// TwinCAT 3 PLC project PMPS
// Title: PMPS
// Company: SLAC - LCLS
// Author: Alex Wallace and contributors
// ProjectVersion: 0.0.0
// Description: Collection of PMPS functionality for LCLS PLCs
// ProgramVersion: 3.1.4023.0
// CompilerDefines: L
// libraries:
//   LCLS General, * (SLAC)
//   Tc2_MC2, * (Beckhoff Automation GmbH)
//   Tc2_Standard, * (Beckhoff Automation GmbH)
//   Tc2_System, * (Beckhoff Automation GmbH)
//   Tc2_Utilities, * (Beckhoff Automation GmbH)
//   Tc3_JsonXml, * (Beckhoff Automation GmbH)
//   Tc3_Module, * (Beckhoff Automation GmbH)
//   TcUnit,1.2.0.0,www.tcunit.org
// project tree:
//   AncillaryComponents/ FB_JsonDocToSafeBP.TcPOU, FB_JsonFileToJsonDoc.TcPOU (not stored), FB_TempSensor_FFO.TcPOU (not stored), FB_PressSensor_FFO.TcPOU (not stored)
//   DUTs/InternalDUT/ E_MPSBeamRates.TcDUT (not stored), E_MPSBeamClasses.TcDUT (not stored), K_Apertures.TcDUT (not stored), K_Attenuators.TcDUT (not stored), K_Stopper.TcDUT, L_Apertures.TcDUT (not stored), L_Attenuators.TcDUT (not stored), L_Stopper.TcDUT (not stored), ST_AttenuatorStatus.TcDUT (not stored), ST_BP_ArbInternal.TcDUT (not stored), ST_FF.TcDUT (not stored), ST_FFInfo.TcDUT (not stored), ST_FFOverride.TcDUT (not stored), ST_PMPS_Aperture.TcDUT (not stored), ST_PMPS_Attenuator.TcDUT (not stored), T_HashTableEntry.TcDUT (not stored)
//   DUTs/ PMPS_CODES.TcDUT (not stored), ST_DeviceState.TcDUT (not stored), ST_DeviceStateExt.TcDUT (not stored), ST_DeviceStateTable.TcDUT (not stored)
//   DUTs/UserDUT/ E_BridgeLinkStatus.TcDUT (not stored), E_BridgeStatus.TcDUT (not stored), E_DataStatus.TcDUT (not stored), E_EcCommState.TcDUT (not stored), ST_ReactiveParams.TcDUT (not stored), ST_BeamParams.TcDUT (not stored), ST_DbStateParams.TcDUT (not stored), ST_Device.TcDUT (not stored)
//   GVLs/ PMPS_GVL.TcGVL (not stored), PMPS_PARAM.TcGVL, PMPS_TOOLS.TcGVL (not stored)
//   HelperFunctions/ FB_DummyHA.TcPOU (not stored), FB_DummyArbIO.TcPOU (not stored), F_BPWithID.TcPOU (not stored), F_DifferentBeamParams.TcPOU (not stored), F_eVExcludeRange.TcPOU (not stored), F_eVIncludeRange.TcPOU (not stored), F_eVRangeCalculator.TcPOU (not stored), F_eVWithinSpec.TcPOU (not stored), F_InitTestBP.TcPOU (not stored), F_SafeBPCompare.TcPOU (not stored), F_SafeBPCompare0Rate.TcPOU (not stored), F_SetBeamParams.TcPOU (not stored), F_SetGoodAttStatus.TcPOU (not stored), F_SetStateParams.TcPOU (not stored), F_PMPS_JSON.TcPOU (not stored), F_ValidReqID.TcPOU (not stored), PE_Ranges.TcPOU (not stored), F_AttenuatorOK.TcPOU (not stored)
//   HelperFunctions/TypeTranslators/ APT_TO_IO.TcPOU (not stored), ATT_TO_IO.TcPOU (not stored), BP_TO_IO.TcPOU (not stored), F_DeviceState_To_DeviceStateExt.TcPOU (not stored), IO_TO_APT.TcPOU (not stored), IO_TO_ATT.TcPOU (not stored), IO_TO_BP.TcPOU (not stored)
//   ImplicitChecks/ CheckBounds.TcPOU (not stored), CheckDivDInt.TcPOU (not stored), CheckDivLInt.TcPOU (not stored), CheckDivLReal.TcPOU (not stored), CheckDivReal.TcPOU (not stored), CheckLRangeSigned.TcPOU (not stored), CheckLRangeUnsigned.TcPOU (not stored), CheckPointer.TcPOU (not stored), CheckRangeSigned.TcPOU (not stored), CheckRangeUnsigned.TcPOU (not stored)
//   / MAIN.TcPOU (not stored), PlcTask.TcTTO (not stored)
//   MajorComponents/Arbiter/ FB_VetoArbiter.TcPOU (not stored), FB_Arbiter.TcPOU (not stored), FB_BeamParamAssertionPool.TcPOU (not stored)
//   MajorComponents/BPTM/ BeamParameterTransitionManager.TcPOU (not stored), E_BPTMState.TcDUT (not stored)
//   MajorComponents/ FB_BPControlDevice.TcPOU (not stored), FB_RateFromEPICS.TcPOU (not stored), FB_BeamClassFromEPICS.TcPOU (not stored), I_LowerAuthority.TcIO (not stored), I_UndulatorComplex.TcIO (not stored), FB_BPRequestor.TcPOU (not stored), FB_LinearDeviceStateTable.TcPOU (not stored), FB_LinearGovernor.TcPOU (not stored), I_HigherAuthority.TcIO (not stored)
//   MajorComponents/PhotonEnergyInterface/ FB_AcceleratorLinks.TcPOU (not stored), FB_Hgvpu.TcPOU (not stored), FB_LPhotonEnergy.TcPOU (not stored), FB_KPhotonEnergy.TcPOU (not stored), FB_PhotonEnergy.TcPOU (not stored), FB_SXU.TcPOU, FB_UndulatorSegment.TcPOU (not stored), F_CalculatePhotonEnergy.TcPOU (not stored)
//   MajorComponents/FastFaults/ FB_FastFault.TcPOU (not stored), FB_HardwareFFOutput.TcPOU
//   MajorComponents/InterPlcComm/ FB_ArbiterToSubSys_IO.TcPOU, FB_BridgeDiagnostics.TcPOU (not stored), FB_SubSysToArbiter_IO.TcPOU (not stored)
//   MajorComponents/InterPlcComm/Sanitization/ I_FallibleLreal.TcIO (not stored), FB_FallibleRealFromEtherCAT.TcPOU (not stored)
//   MajorComponents/PMPS_MPS_Interface/ FB_BeamClassOutputs.TcPOU (not stored), FB_BeamClassOutputs_BCD.TcPOU (not stored), FB_CTLS_Outputs.TcPOU (not stored), FB_MachineModeFromEPICS.TcPOU (not stored), FB_PhotonEnergyWatcher.TcPOU (not stored), FB_BeamClassWatcher.TcPOU (not stored)
//   MajorComponents/SimulationFB/ FB_eVSimulator.TcPOU (not stored), FB_MachineSimulator.TcPOU (not stored)
//   MajorComponents/Stoppers/ FB_KStopper.TcPOU (not stored), FB_KVetoDevice.TcPOU (not stored), FB_LVetoDevice.TcPOU (not stored), FB_LStopper.TcPOU (not stored), FB_StopperWatcher.TcPOU (not stored), FB_VetoDevice.TcPOU (not stored)
//   TestComponents/DUT/ E_ArbDosTestStates.TcDUT (not stored), E_BPTMTestStates.TcDUT (not stored)
//   TestComponents/ FB_Arbiter_Test.TcPOU (not stored), FB_VetoArbiter_Test.TcPOU (not stored), FB_AttenuatorSimulator.TcPOU (not stored), FB_BPTM_Test.TcPOU (not stored), FB_ArbToSubsys_Test.TcPOU (not stored), FB_DiffBP_Test.TcPOU (not stored), FB_SubsysToArb_Test.TcPOU (not stored), FB_evRangeCalculator_Test.TcPOU (not stored), FB_eVWithinSpec_Test.TcPOU (not stored), FB_FastFault_Test.TcPOU (not stored), FB_PhotonEnergyWatcher_Test.TcPOU (not stored), FB_SafeBPCompare_Test.TcPOU (not stored), FB_SolidAttenuator.TcPOU (not stored) (excluded from build)

// ---- DUTs/InternalDUT/K_Stopper.TcDUT
{attribute 'qualified_only'}
{attribute 'strict'}
TYPE K_Stopper :
(
    ST3K4 := 1, // TMO PPS stopper in
    ST1K2 := 2, // RIX PPS stopper in
    MR1K1_IN := 3, // Monochromator focus optic vertical state
    MR1K1_OUT := 4, // Monochromator focus optic vertical state
    MR1K3_IN := 5, // TXI MR1K3 Offset Mirror horizontal state
    MR1K3_OUT := 6, // TXI MR1K3 Offset Mirror horizontal state
    ST4K4 := 7, //TMO ST4K4 Photon Terminator In Limit Switch
    ST1K0 := 8, //Test Photon Stopper in the FEE
    ST1K3 :=9, //TXI Kline PPS stopper in
    MR2K3_IN := 10, // TXI MR2K3 Offset Mirror state
    MR2K3_OUT := 11, // TXI MR2K3 Offset Mirror horizontal state
    DEFAULT := PMPS_GVL.MAX_VETO_DEVICES // DO NOT USE FOR ANYTHING
);
END_TYPE

// ---- GVLs/PMPS_PARAM.TcGVL
{attribute 'qualified_only'}
VAR_GLOBAL CONSTANT
    MAX_FAST_FAULTS	:	UINT := 50; // Max fast faults for an FFO
    MAX_ASSERTIONS    :    UDINT := 20; //Maximum number of BP requests in the arbiter
    TRANS_MARGIN : REAL := REAL#0.05; // Allowed % margin above requested transmission level in SafeBPCompare (0.0500 = 5deci% default). Note: change this value if scaling factor changes.
END_VAR

// ---- AncillaryComponents/FB_JsonDocToSafeBP.TcPOU
FUNCTION_BLOCK FB_JsonDocToSafeBP
VAR_INPUT
	bExecute             : BOOL; //Rising Edge
	jsonDoc 		: SJsonValue;
	sDeviceName : STRING;
END_VAR
VAR_OUTPUT
	bHasDevice		: BOOL;
	bHasAllStates		: BOOL;
	bHasAllParameters :BOOL := TRUE;
	bBusy                : BOOL;
    bError               : BOOL;
    nErrId               : UDINT;
	sErrMsg				 :STRING;
END_VAR
VAR_IN_OUT
	arrStates: ARRAY[*] OF ST_DbStateParams;
	io_fbFFHWO    :    FB_HardwareFFOutput;
END_VAR
VAR
	(* JSON *)
	fbJson 			: FB_JsonDomParser;
	jsonProp		: SJsonValue;
	jsonValue		: SJsonValue;
	jsonParam		: SJsonValue;
	jsonnTran      : SJsonValue;
	jsonnRate      : SJsonValue;
	Step: INT;
	index: DINT;
	nStateCount:DINT;
    RisingEdge           : R_TRIG;

	(*Logger*)
	tNewMessage : R_TRIG;
    fbLogger : FB_LogMessage := (eSubsystem:=E_SubSystem.MPS, nMinTimeViolationAcceptable:=10);	
	(*FFO*)
	FFO    :    FB_FastFault :=(
        i_Desc := 'Fault occurs when there is an error loading safe beam parameters from json file',
        i_TypeCode := 16#FF13);
	sbuffReadSmall: INT;
END_VAR

(* Retrieve JSON content *)
RisingEdge(CLK:=bExecute); 

CASE Step OF 
    0:     (* Idle state *) 
          IF RisingEdge.Q THEN 
               bBusy := TRUE; 
               bError:= FALSE; 
               nErrId:=0; 
			   sErrMsg :='';
               Step := 20; 
			   fbLogger(sMsg:='Start Parsing Json DOC.', eSevr:=TcEventSeverity.Info);
          END_IF 
	
	 20: (*Find the Device Name*)  
		bHasDevice := fbJson.HasMember(jsonDoc, sDeviceName);
		IF (bHasDevice) THEN
			jsonProp := fbJson.FindMember(jsonDoc, sDeviceName);
			IF jsonProp <> 0 THEN	
				Step := Step+1;
				ELSE
					Step := 900 + Step;
					nErrId := Step; 
					bError := TRUE; 
					sErrMsg:=  CONCAT('Error device name not found in Json File : ',sDeviceName);
				END_IF
		ELSE
			Step := 900 + Step;
			nErrId := Step; 
			bError := TRUE; 
			sErrMsg:=  CONCAT('Error device name not found in Json File : ',sDeviceName);		
		END_IF
		
	 21: (*Check device States in DOM*)
	 		nStateCount :=0;
	 		FOR Index:=LOWER_BOUND(arrStates,1) TO UPPER_BOUND(arrStates,1) BY 1 DO
				  IF NOT ((arrStates[Index].sPmpsState= '') OR (arrStates[Index].sPmpsState= 'Invalid')) THEN
					  IF NOT (fbJson.HasMember(jsonProp, arrStates[Index].sPmpsState)) THEN
							  Step := 900+ Step;
							  nErrId := Step; 
							  bError := TRUE; 
							  sErrMsg:= CONCAT('Error loading device state in Json File : ',arrStates[Index].sPmpsState);
							  fbLogger(sMsg:= sErrMsg, eSevr:=TcEventSeverity.Critical);
							  EXIT;
					    ELSE 
							nStateCount :=nStateCount+1;
					  END_IF
				   ELSE   
					   bHasAllStates :=TRUE;
					   EXIT;
				  END_IF
		    END_FOR

		   Step := Step+1;
			
	 22: //MAke sure state array input has State name data
		  IF (nStateCount =0) THEN
			  bHasAllStates :=FALSE;
			  Step := 900+ Step;
			  nErrId := Step; 
			  bError := TRUE; 
			  sErrMsg:= CONCAT('Error Input State array is empty : ',sDeviceName);				  
		 ELSE 
			 Step := Step+1;		 
		 END_IF;

	 23:  (*loop Device State Arrays to find load all States BP*)
	      FOR Index:=LOWER_BOUND(arrStates,1) TO UPPER_BOUND(arrStates,1) BY 1 DO
			  IF NOT (arrStates[Index].sPmpsState= '') THEN
				  IF(NOT M_LoadSafeBP(arrStates[Index].sPmpsState, Index)) THEN
					  Step := 900+ Step;
					  fbLogger.sMsg := CONCAT('Error Parsing beam parameters - Device/States: ', arrStates[Index].sPmpsState);
					  fbLogger(sMsg:= sErrMsg, eSevr:=TcEventSeverity.Critical);
				  END_IF
			   ELSE 
					EXIT;
			   END_IF
		  END_FOR
		  IF (bHasAllParameters) THEN Step := 30;
			  ELSE Step := 900+ Step;
		  END_IF
		  
	 30: (*ALL good here*)
	 	fbLogger.sMsg := CONCAT('Complete Parsing Json Doc. Device: ', sDeviceName);
		fbLogger.sMsg := CONCAT(fbLogger.sMsg ,' - States Count: ');
		fbLogger.sMsg := CONCAT(fbLogger.sMsg ,TO_STRING(nStateCount));
	  	fbLogger(eSevr:=TcEventSeverity.Info);
	 	bExecute:= FALSE;
	    bBusy:=FALSE;
		Step := 0;
		FFO.i_xOK := TRUE;
END_CASE


//Fault in error state
IF(Step>=900) THEN
	FFO.i_xOK := FALSE;
	Step:=0;
END_IF
ACT_FFO();
ACT_LOGGER();

ACTION ACT_FFO:
(*FAST FAULT*)
FFO(i_xOK := ,
    i_xReset := ,
	i_xAutoReset :=TRUE,
	i_DevName := sDeviceName,
    io_fbFFHWO := io_fbFFHWO);
END_ACTION

ACTION ACT_Logger:
// Log valve open
tNewMessage(CLK:= NOT(FbLogger.sMsg = sErrMsg) AND NOT (sErrMsg =''));
IF tNewMessage.Q THEN fbLogger(sMsg:= sErrMsg, eSevr:=TcEventSeverity.Critical); END_IF
END_ACTION

METHOD M_LoadSafeBP : BOOL
VAR_INPUT
	sStateName : STRING;
	Index:DINT;
END_VAR
VAR
	//bHasAllParameters : BOOL := TRUE;
	sAperture:STRING;
	nAperture:INT := -1;
	sEV:STRING;
	sBC:STRING;
	nIndex:INT;
END_VAR
bHasAllParameters :=  fbJson.HasMember(jsonProp, sStateName);
jsonValue := fbJson.FindMember(jsonProp, sStateName);
IF bHasAllParameters THEN
	//nTran
	bHasAllParameters R= NOT fbJson.HasMember(jsonValue, 'nTran');
	IF (NOT bHasAllParameters) THEN fbLogger(sMsg:= 'Error Loading nTran', eSevr:=TcEventSeverity.Critical); END_IF
	jsonnTran := fbJson.FindMember(jsonValue, 'nTran');
	arrStates[Index].stBeamParams.nTran := TO_REAL(fbJson.GetString(jsonnTran));
	
	//nRate
	bHasAllParameters R= NOT fbJson.HasMember(jsonValue, 'nRate');
	IF (NOT bHasAllParameters) THEN fbLogger(sMsg:= 'Error Loading nRate', eSevr:=TcEventSeverity.Critical); END_IF
	jsonnRate := fbJson.FindMember(jsonValue, 'nRate');
	arrStates[Index].stBeamParams.nRate:= TO_UDINT(fbJson.GetString(jsonnRate));
	
	//neVRange
	bHasAllParameters R= NOT fbJson.HasMember(jsonValue, 'neVRange');
	jsonParam := fbJson.FindMember(jsonValue, 'neVRange');
	sEV:=(fbJson.GetString(jsonParam));
	bHasAllParameters R= NOT (LEN(sEV)=32);
	This^.arrStates[Index].stBeamParams.neVRange :=0;
	IF (NOT bHasAllParameters) THEN 
		fbLogger(sMsg:= 'Error Loading eVRange', eSevr:=TcEventSeverity.Critical); 
		ELSE
			FOR nIndex := 0 TO PMPS_GVL.g_cBoundaries BY 1 DO
				This^.arrStates[Index].stBeamParams.neVRange := SHL(This^.arrStates[Index].stBeamParams.neVRange,1);
				This^.arrStates[Index].stBeamParams.neVRange := This^.arrStates[Index].stBeamParams.neVRange+HEXASCNIBBLE_TO_BYTE(sEV[nIndex]);
			END_FOR
	END_IF
	
	//nBeamClassRange
	bHasAllParameters R= NOT fbJson.HasMember(jsonValue, 'nBeamClassRange');
	jsonParam := fbJson.FindMember(jsonValue, 'nBeamClassRange');
	sBC:=(fbJson.GetString(jsonParam));
	bHasAllParameters R= NOT (LEN(sBC)=15);
	arrStates[Index].stBeamParams.nBCRange :=0;
	IF (NOT bHasAllParameters) THEN 
			fbLogger(sMsg:= 'Error Loading Beam Class Range. Make sure Bitmask is equal than 15 bits.', eSevr:=TcEventSeverity.Critical);
	ELSE
		FOR nIndex := 0 TO 14 BY 1 DO
			arrStates[Index].stBeamParams.nBCRange := SHL(arrStates[Index].stBeamParams.nBCRange,1);
			arrStates[Index].stBeamParams.nBCRange := arrStates[Index].stBeamParams.nBCRange+HEXASCNIBBLE_TO_BYTE(sBC[nIndex]);
		END_FOR
	 END_IF
	
	//ApertureName and Values
	bHasAllParameters R= NOT fbJson.HasMember(jsonValue, 'ap_name');
	jsonParam := fbJson.FindMember(jsonValue, 'ap_name');
	sAperture := fbJson.GetString(jsonParam);
{IF defined (L)}
	IF ('SL1L0' = sAperture) THEN nAperture := L_Apertures.SL1L0;
	ELSIF ('SL2L0' = sAperture) THEN nAperture := L_Apertures.SL2L0; 
	END_IF
{ELSIF defined (K)} // Attribute 'to_string' only build 4024 TO_STRING(PMPS.K_Apertures.SL1K0) - need another non hardcoded way
	IF ('SL1K0' = sAperture) THEN nAperture := K_Apertures.SL1K0;
	ELSIF ('SL2K0' = sAperture) THEN nAperture := K_Apertures.SL2K0;
	END_IF
{END_IF}
	IF (nAperture>-1) THEN	
		//Gap Height
		bHasAllParameters R= NOT fbJson.HasMember(jsonValue, 'ap_ygap');
		jsonParam := fbJson.FindMember(jsonValue, 'ap_ygap');
		arrStates[Index].stBeamParams.astApertures[nAperture].Height := TO_REAL(fbJson.GetString(jsonParam));
		
		//Gap Width
		bHasAllParameters R= NOT fbJson.HasMember(jsonValue, 'ap_xgap');
		jsonParam := fbJson.FindMember(jsonValue, 'ap_xgap');
		arrStates[Index].stBeamParams.astApertures[nAperture].Width := TO_REAL(fbJson.GetString(jsonParam));

		IF (NOT bHasAllParameters) THEN fbLogger(sMsg:= 'Error Loading aperture gap', eSevr:=TcEventSeverity.Critical); END_IF	
	END_IF
	
	//Read Transition ID for the State
	bHasAllParameters R= NOT fbJson.HasMember(jsonValue, 'id');
	jsonParam := fbJson.FindMember(jsonValue, 'id');
	IF (NOT bHasAllParameters) THEN fbLogger(sMsg:= 'Error Loading Assertion ID', eSevr:=TcEventSeverity.Critical); END_IF
	arrStates[Index].nRequestAssertionID := TO_UDINT(fbJson.GetInt(jsonParam));
	
	//Set to True to indicate this state has been initialized
	arrStates[Index].bBeamParamsLoaded := bHasAllParameters;
END_IF

IF NOT(	bHasAllParameters) THEN
	nErrId := 900+Step; 
    bError := TRUE; 
	sErrMsg:= CONCAT('Error loading BP Data - Device-State: ',sStateName); 	
	fbLogger(sMsg:= sErrMsg, eSevr:=TcEventSeverity.Critical);
END_IF

M_LoadSafeBP:=bHasAllParameters;



//TODO
//ADD the rest of the BP
END_METHOD

END_FUNCTION_BLOCK

// ---- MajorComponents/FastFaults/FB_HardwareFFOutput.TcPOU
{attribute 'reflection'}
{attribute 'no_check'}
FUNCTION_BLOCK FB_HardwareFFOutput
VAR CONSTANT
    FF_ARRAY_UPPER_BOUND : UINT := PMPS_PARAM.MAX_FAST_FAULTS;
END_VAR
VAR_INPUT
	//FF_ARRAY_UPPER_BOUND : UINT := PMPS_PARAM.MAX_FAST_FAULTS;
    {attribute 'pytmc' := '
        pv: ClearFault
        io: o
        field: DESC Might be overidden by PLC writes
     '}
    i_xReset    :    BOOL;
    {attribute 'pytmc' := '
        pv: EnableVeto
        io: o
     '}
    i_xVeto    :    BOOL;
    bAutoReset : BOOL := FALSE; // Set true for the FFO to automatically permit beam again after all fast faults are cleared
    i_sNetID : T_AmsNetID:=''; //Set to the Arbiter AmsNetID to be used for the synchronisation. An empty string means the system will sue local time
END_VAR
VAR_OUTPUT
    {attribute 'pytmc' := '
        pv: FaultHWO
        io: i
        field: DESC Hardware Output Status
     '}
    q_xFastFaultOut    AT %Q*    :    BOOL;
    q_xValidSyncTime : BOOL;// system time bValid output True when sync is successful
END_VAR
VAR_IN_OUT
    
END_VAR
VAR
    {attribute 'pytmc' := '
        pv: FF
     '}
    astFF : ARRAY[1..FF_ARRAY_UPPER_BOUND] OF ST_FF;
	{attribute 'pytmc' := '
        pv: RegistrationFailure
        io: io
     '}
    xFastFaultRegFail  :   BOOL := FALSE; // Set true if a fast fault fails to register. Holds beam off.
    tFFRegFail : F_TRIG;

    {attribute 'instance-path'}
    {attribute 'noinit'}
    sPath    :    T_MaxString;

    {attribute 'pytmc' := '
        pv: OK
        io: i
     '}
    xOK    :    BOOL:= TRUE; // Current internal state of FFO, indicates if FFO will accept a reset

    rtReset    :    R_TRIG;
    rtResetandOK : R_TRIG;

    nIndex    :    UINT := 1;

    IdxOK: BOOL;

    fbTime : FB_LocalSystemTime := ( bEnable := TRUE, dwCycle := 1 ); //Get current system time, used for override
    fbTime_to_UTC: FB_TzSpecificLocalTimeToSystemTime;
    fbGetTimeZone: FB_GetTimeZoneInformation;
    fbJson : FB_JsonSaxWriter;
    pmpsTypeCode : UDINT := 0; // shows up in json as pmps_typecode
    fbLogger : FB_LogMessage := (
        eSevr := TcEventSeverity.Critical,
        eSubsystem := E_Subsystem.MPS,
        nMinTimeViolationAcceptable := FF_ARRAY_UPPER_BOUND);

END_VAR

// <TODO> latch off beam if DI card status goes bad

ACTION EvaluateOutput:

////////////////////////////////////////////////////////////////
// Critical code. Do not touch unless you know what you're doing
////////////////////////////////////////////////////////////////

//<TODO> add diagnostic for success or failure of reset
rtReset(CLK:=i_xReset);
rtResetandOK(CLK:=(rtReset.Q OR bAutoReset) AND xOK);

q_xFastFaultOut S= rtResetandOK.Q;
q_xFastFaultOut R= (NOT xOK OR xFastFaultRegFail);

//Reset OK for next cycle
xOK := True;

////////////////////////////////////////////////////////////////
END_ACTION

{attribute 'no_check'}
METHOD EvaluateOverrides : BOOL
VAR_INPUT
END_VAR
VAR
    FF : REFERENCE TO ST_FF;
    EvalIdx: DINT := 1;
END_VAR
VAR CONSTANT
    MaxTime : DINT:= 4294080;(*49.7 days*)
END_VAR
//Get local System Time
fbTime(sNetID:=i_sNetID);
//Get Time Zone
fbGetTimeZone(sNetID:=i_sNetID,bExecute:=TRUE,tTimeout:=T#10S);
//change local time to UTC to be compatible with unix time epoch widget
fbTime_to_UTC(in:= fbTime.systemTime , tzInfo:=fbGetTimeZone.tzInfo);
q_xValidSyncTime := fbTime.bValid AND NOT fbGetTimeZone.bError;

FOR EvalIdx := 1 TO FF_ARRAY_UPPER_BOUND DO

    FF REF= astFF[EvalIdx];

    IF NOT FF.Info.InUse THEN
        CONTINUE;
    ELSE
        // Veto timer
        IF FF.Ovrd.Deactivate THEN
            FF.Ovrd.Timer.PT := T#0s; // Only needs to be set zero for one cycle
        ELSIF FF.Ovrd.Activate THEN
            FF.Ovrd.StartDT:= TO_DINT(TO_DT(SystemTime_TO_DT(fbTime_to_UTC.out)));
            IF (FF.Ovrd.StartDT < FF.Ovrd.Expiration) THEN
                FF.Ovrd.Expiration:= LIMIT(0,FF.Ovrd.Expiration, FF.Ovrd.StartDT+MaxTime );
                   FF.Ovrd.Timer.PT := TO_DT(FF.Ovrd.Expiration)- SystemTime_TO_DT(fbTime_to_UTC.out);
            END_IF
        END_IF

        // UDINT conversions for ESS module compatibility.
        FF.Ovrd.Timer(
            IN := FF.Ovrd.Activate, // Rising edge activated
            Q => FF.Ovrd.Active);

        FF.Ovrd.tOvrdActivate(CLK:=FF.Ovrd.Active);
        FF.Ovrd.OvrdActLogAck S= FF.Ovrd.tOvrdActivate.Q;

        FF.Ovrd.tOvrdExpiring(CLK:=FF.Ovrd.Active);
        FF.Ovrd.OvrdExpLogAck S= FF.Ovrd.tOvrdExpiring.Q;

        FF.Ovrd.ElapsedTime := TIME_TO_UDINT(FF.Ovrd.Timer.ET);

        FF.Ovrd.RemainingTime := MAX(0, TO_DINT(FF.Ovrd.Timer.PT) - FF.Ovrd.ElapsedTime);

        // Clear pushbuttons
        FF.Ovrd.Activate := FALSE;
        FF.Ovrd.Deactivate := FALSE;

    END_IF
END_FOR
END_METHOD

{attribute 'obsolete' := 'Use EvaluateOverrides instead.'}
METHOD EvaluateVetos : BOOL
VAR_INPUT
END_VAR
END_METHOD

ACTION Execute:
EvaluateOverrides();
EvaluateOutput();
ExecuteLogging();
END_ACTION

{attribute 'no_check'}
METHOD ExecuteLogging : BOOL
VAR_INPUT
END_VAR
VAR
    FF : REFERENCE TO ST_FF;
    logIdx : DINT := 1;
END_VAR
VAR_INST
    HelloTimer : TOF := ( PT:=T#24h );
END_VAR

FOR logIdx := 1 to FF_ARRAY_UPPER_BOUND do

    FF REF= astFF[logIdx];

    IF NOT FF.Info.InUse THEN
        CONTINUE;
    ELSE
        IF FF.FaultAck THEN

            pmpsTypeCode := 1;
            FormulateLogJson(FF);
            fbLogger(sMsg := 'Fault, beam off', eSevr:=TcEventSeverity.Critical);

            FF.FaultAck := FALSE;
        END_IF

        IF FF.Ovrd.OvrdActLogAck THEN

            pmpsTypeCode := 2;
            FormulateLogJson(FF);

            fbLogger(sMsg := 'Override activated', eSevr:=TcEventSeverity.Warning);

            FF.Ovrd.OvrdActLogAck := FALSE;
        END_IF

        IF FF.Ovrd.OvrdExpLogAck THEN

            pmpsTypeCode := 3;
            FormulateLogJson(FF);

            fbLogger(sMsg := 'Override released', eSevr:=TcEventSeverity.Warning);

            FF.Ovrd.OvrdExpLogAck := FALSE;
        END_IF

        IF FF.ClearAck THEN

            pmpsTypeCode := 8;
            FormulateLogJson(FF);

            fbLogger(sMsg := 'Fault cleared', eSevr:=TcEventSeverity.Info);

            FF.ClearAck := FALSE;
        END_IF


    END_IF
END_FOR

// Log registration fault cleared
tFFRegFail(CLK:=xFastFaultRegFail);
IF tFFRegFail.Q THEN
    fbJson.StartObject();
    fbJson.AddKey('pmps_typecode');
    fbJson.AddUdint(5);
    fbJson.AddKey('pmps_path');
    fbJson.AddString(sPath);
    fbJson.EndObject();
    fbJson.CopyDocument(pDoc:=fbLogger.sJson, SIZEOF(fbLogger.sJson));
    fbLogger(sMsg := 'Fast fault registration failure cleared. This may be bad as a fast fault could go unoticed.',
        eSevr:=TcEventSeverity.Warning);
END_IF

// Say hello
HelloTimer.IN := NOT HelloTimer.Q;
HelloTimer();
IF HelloTimer.IN THEN
    pmpsTypeCode := 10;
    FormulateLogJson(FF);
    fbLogger(eSubsystem:=E_Subsystem.NILVALUE,
        eSevr := TcEventSeverity.Info,
        sMsg := 'FFO is alive');
    fbLogger.eSubsystem := E_Subsystem.MPS;
END_IF
END_METHOD

ACTION ExecuteNoLog:
EvaluateOverrides();
EvaluateOutput();
//ExecuteLogging();
END_ACTION

METHOD INTERNAL FormulateLogJson : STRING
VAR_INPUT
    FF : ST_FF;
END_VAR
fbJson.StartObject();
fbJson.AddKey('pmps_typecode');
fbJson.AddUdint(pmpsTypeCode);
fbJson.AddKey('pmps_path');
fbJson.AddString(FF.Info.sPath);
fbJson.AddKey('pmps_device_name');
fbJson.AddString(FF.Info.DevName);
fbJson.EndObject();
fbLogger.sJson := fbJson.GetDocument();
fbJson.ResetDocument();
END_METHOD

{attribute 'no_check'}
METHOD INTERNAL IdxCheckIn : BOOL
VAR_INPUT
    Idx : DINT;
    OK : BOOL;
    Reset : BOOL;
END_VAR
VAR
    stFF : ST_FF;
    BeamPermitted : BOOL;
END_VAR
Idx := LIMIT(1,Idx,FF_ARRAY_UPPER_BOUND);
stFF := THIS^.astFF[Idx];

// Updating internal fault state
stFF.OK := OK;

// Reset and latching logic
stFF.rtReset(CLK:=stFF.Reset (*epics*) OR Reset (*from other PLC logic *) );
stFF.Reset R= stFF.rtReset.Q;
stFF.bsFF(SET := stFF.rtReset.Q OR stFF.Info.AutoReset, RESET1:= NOT OK);

BeamPermitted := stFF.bsFF.Q1 OR stFF.Ovrd.Active OR (i_xVeto AND stFF.Info.Vetoable);

// Fault generation
IF NOT BeamPermitted THEN
    THIS^.xOK := FALSE; //Very clever, thanks Zach!
END_IF

// Fast fault accumulation
stFF.ftCountFault(CLK:=stFF.bsFF.Q1);
IF stFF.ftCountFault.Q THEN PMPS_GVL.AccumulatedFF := PMPS_GVL.AccumulatedFF + 1; END_IF

//Clear pushbuttons
stFF.Reset := FALSE;

// Log when this fault faults
stFF.FaultAck S= stFF.BeamPermitted AND NOT BeamPermitted;

// Log when this fault has cleared
stFF.ClearAck S= BeamPermitted AND NOT stFF.BeamPermitted;

stFF.BeamPermitted := BeamPermitted;

// Copy state back to ff struct
THIS^.astFF[Idx] := stFF;
END_METHOD

{attribute 'no_check'}
METHOD INTERNAL Register : BOOL
VAR_INPUT
    stFFInfo : ST_FFInfo := (
        sPath := '',
        Desc := '',
        TypeCode := 16#00,
        DevName := ''); // Fast fault information

END_VAR
VAR_OUTPUT
    FFOName : T_MaxString;
    Idx : UINT;
END_VAR
VAR
END_VAR
FFOName := THIS^.sPath;
Idx := THIS^.nIndex;

IF THIS^.nIndex <= FF_ARRAY_UPPER_BOUND THEN

    THIS^.astFF[MIN(THIS^.nIndex,FF_ARRAY_UPPER_BOUND)].Info:=stFFInfo;
	
    THIS^.nIndex := THIS^.nIndex + 1;

    Register := TRUE; // Add successful
ELSE
    fbJson.StartObject();
    fbJson.AddKey('pmps_typecode');
    fbJson.AddUdint(4);
    fbJson.AddKey('pmps_path');
    fbJson.AddString(stFFInfo.sPath);
    fbJson.AddKey('pmps_device_name');
    fbJson.AddString(stFFInfo.DevName);
    fbJson.EndObject();
    fbLogger.sJson := fbJson.GetDocument();
    fbJson.ResetDocument();
    fbLogger(sMsg:='Fast fault registration failed. Too many fast faults on this FFO.',
        eSevr:=TcEventSeverity.Warning,
        eSubsystem:=E_Subsystem.MPS);
    xFastFaultRegFail := TRUE;
    Register := FALSE; // Failed to add name to list
END_IF
END_METHOD

END_FUNCTION_BLOCK

// ---- MajorComponents/PhotonEnergyInterface/FB_SXU.TcPOU
FUNCTION_BLOCK FB_SXU IMPLEMENTS I_UndulatorComplex
VAR_INPUT
    fbElectronEnergy : REFERENCE TO FB_LREALFromEPICS;
END_VAR

VAR_OUTPUT
    {attribute 'pytmc' := '
        pv: CurrentPhotonEnergy
        io: i
        field: DESC Calculated current photon energy
        field: PREC 3
        field: EGU eV
    '}
    fCurrentPhotonEnergy : LREAL;
    {attribute 'pytmc' := '
        pv: TargetPhotonEnergy
        io: i
        field: DESC Calculated desired photon energy
        field: PREC 3
        field: EGU eV
    '}
    fTargetPhotonEnergy : LREAL;
        {attribute 'pytmc' := '
        pv: SeedUndulatorNumber
        io: i
        field: DESC Seed undulator number
    '}
    nSeedUndulator : UDINT; // Set to zero when no undulators are active
    {attribute 'pytmc' := '
        pv: TargetSeedUndulatorNumber
        io: i
        field: DESC Seed undulator number for target K
    '}
    nTargetSeedUndulator : UDINT; // Set to zero when no undulators are active
END_VAR



VAR
    // From lcls-srv01: grep -e KDes  /u1/lcls/epics/ioc/data/sioc-unds-uc*/iocInfo/IOC.pvlist |sort

    {attribute 'pytmc' := 'pv: 19; link: 1950:'}
    fbSegment_19 : FB_UndulatorSegment;

    {attribute 'pytmc' := 'pv: 20; link: 2050:'}
    fbSegment_20 : FB_UndulatorSegment;

    {attribute 'pytmc' := 'pv: 21; link: 2150:'}
    fbSegment_21 : FB_UndulatorSegment;

    {attribute 'pytmc' := 'pv: 22; link: 2250:'}
    fbSegment_22 : FB_UndulatorSegment;

    {attribute 'pytmc' := 'pv: 23; link: 2350:'}
    fbSegment_23 : FB_UndulatorSegment;

    {attribute 'pytmc' := 'pv: 24; link: 2450:'}
    fbSegment_24 : FB_UndulatorSegment;

    {attribute 'pytmc' := 'pv: 25; link: 2550:'}
    fbSegment_25 : FB_UndulatorSegment;

    {attribute 'pytmc' := 'pv: 26; link: 2650:'}
    fbSegment_26 : FB_UndulatorSegment;

    {attribute 'pytmc' := 'pv: 27; link: 2750:'}
    fbSegment_27 : FB_UndulatorSegment;

    {attribute 'pytmc' := 'pv: 28; link: 2850:'}
    fbSegment_28 : FB_UndulatorSegment;

    {attribute 'pytmc' := 'pv: 29; link: 2950:'}
    fbSegment_29 : FB_UndulatorSegment;

    {attribute 'pytmc' := 'pv: 30; link: 3050:'}
    fbSegment_30 : FB_UndulatorSegment;

    {attribute 'pytmc' := 'pv: 31; link: 3150:'}
    fbSegment_31 : FB_UndulatorSegment;

    {attribute 'pytmc' := 'pv: 32; link: 3250:'}
    fbSegment_32 : FB_UndulatorSegment;

    {attribute 'pytmc' := 'pv: 33; link: 3350:'}
    fbSegment_33 : FB_UndulatorSegment;

    {attribute 'pytmc' := 'pv: 34; link: 3450:'}
    fbSegment_34 : FB_UndulatorSegment;

    {attribute 'pytmc' := 'pv: 36; link: 3650:'}
    fbSegment_36 : FB_UndulatorSegment;

    {attribute 'pytmc' := 'pv: 37; link: 3750:'}
    fbSegment_37 : FB_UndulatorSegment;

    {attribute 'pytmc' := 'pv: 38; link: 3850:'}
    fbSegment_38 : FB_UndulatorSegment;

    {attribute 'pytmc' := 'pv: 39; link: 3950:'}
    fbSegment_39 : FB_UndulatorSegment;

    {attribute 'pytmc' := 'pv: 40; link: 4050:'}
    fbSegment_40 : FB_UndulatorSegment;

    {attribute 'pytmc' := 'pv: 41; link: 4150:'}
    fbSegment_41 : FB_UndulatorSegment;

    {attribute 'pytmc' := 'pv: 42; link: 4250:'}
    fbSegment_42 : FB_UndulatorSegment;

    {attribute 'pytmc' := 'pv: 43; link: 4350:'}
    fbSegment_43 : FB_UndulatorSegment;

    {attribute 'pytmc' := 'pv: 44; link: 4450:'}
    fbSegment_44 : FB_UndulatorSegment;

    {attribute 'pytmc' := 'pv: 45; link: 4550:'}
    fbSegment_45 : FB_UndulatorSegment;

    {attribute 'pytmc' := 'pv: 46; link: 4650:'}
    fbSegment_46 : FB_UndulatorSegment;

    {attribute 'pytmc' := 'pv: 47; link: 4750:'}
    fbSegment_47 : FB_UndulatorSegment;



    fbSegment : ARRAY [iLowBound..iHighBound] OF POINTER TO FB_UndulatorSegment;
    fbCurrentSegment : REFERENCE TO FB_UndulatorSegment;

    iIndex : UDINT;

    bInitialized : BOOL := FALSE;

END_VAR

VAR CONSTANT
    {attribute 'pytmc' := '
        pv: FirstSegment
        io: i'}
    iLowBound  : UDINT := 19;
    {attribute 'pytmc' := '
        pv: LastSegment
         io: i'}
    iHighBound : UDINT := 47;
    {attribute 'pytmc' := '
        pv: Period_Short
        io: i
        field: EGU mm
    '}
    fPeriod_39_mm : LREAL := 39.0;

    {attribute 'pytmc' := '
        pv: Period_Long
        io: i
        field: EGU mm
    '}
    fPeriod_56_mm : LREAL := 56.0;

    {attribute 'pytmc' := '
        pv: LowK
        io: i
    '}
    fLowK : LREAL := 1.52;

    {attribute 'pytmc' := '
        pv: HiK
        io: i
    '}
    fHiK : LREAL := 20;
END_VAR



IF NOT bInitialized THEN
    Init();
END_IF

UndAdrUpdate();

nSeedUndulator := 0;
nTargetSeedUndulator := 0;

FOR iIndex := iLowBound TO iHighBound DO
    IF fbSegment[iIndex] <> 0 THEN
        fbCurrentSegment REF= fbSegment[iIndex]^;
        fbCurrentSegment(fbElectronEnergy:=fbElectronEnergy);
        fbCurrentSegment.fPeriod_mm := fbCurrentSegment.fLambda_U*1000;

        //Mark the seed undulator, first undulator operating within K bounds
        IF fbCurrentSegment.xActive AND nSeedUndulator = 0 THEN
            nSeedUndulator := iIndex;
            fCurrentPhotonEnergy := fbCurrentSegment.fPhotonEnergyAct;
        END_IF

        IF fbCurrentSegment.xTargetActive AND nTargetSeedUndulator = 0 THEN
            nTargetSeedUndulator := iIndex;
            fTargetPhotonEnergy := fbCurrentSegment.fPhotonEnergyDes;
        END_IF
    END_IF
END_FOR

IF nSeedUndulator = 0 THEN
    fCurrentPhotonEnergy := 0;
END_IF

IF nTargetSeedUndulator = 0 THEN
    fTargetPhotonEnergy := 0;
END_IF

ACTION Init:

UndAdrUpdate();

FOR iIndex := iLowBound TO iHighBound DO
        IF fbSegment[iIndex] <> 0 THEN
        fbCurrentSegment REF= fbSegment[iIndex]^;
        fbCurrentSegment.fLowK := fLowK;
        fbCurrentSegment.fHiK := fHiK;
    END_IF
END_FOR
bInitialized := TRUE;
END_ACTION

PROPERTY rCurrentPhotonEnergy : REAL
GET
rCurrentPhotonEnergy := fCurrentPhotonEnergy;
END_GET
END_PROPERTY

PROPERTY rTargetPhotonEnergy : REAL
GET
rTargetPhotonEnergy := fTargetPhotonEnergy;
END_GET
END_PROPERTY

ACTION UndAdrUpdate:
fbSegment[19] := ADR(fbSegment_19);
fbSegment[20] := ADR(fbSegment_20);
fbSegment[21] := ADR(fbSegment_21);
fbSegment[22] := ADR(fbSegment_22);
fbSegment[23] := ADR(fbSegment_23);
fbSegment[24] := ADR(fbSegment_24);
fbSegment[25] := ADR(fbSegment_25);
fbSegment[26] := ADR(fbSegment_26);
fbSegment[27] := ADR(fbSegment_27);
fbSegment[28] := ADR(fbSegment_28);
fbSegment[29] := ADR(fbSegment_29);
fbSegment[30] := ADR(fbSegment_30);
fbSegment[31] := ADR(fbSegment_31);
fbSegment[32] := ADR(fbSegment_32);
fbSegment[33] := ADR(fbSegment_33);
fbSegment[34] := ADR(fbSegment_34);
fbSegment[35] := 0;
fbSegment[36] := ADR(fbSegment_36);
fbSegment[37] := ADR(fbSegment_37);
fbSegment[38] := ADR(fbSegment_38);
fbSegment[39] := ADR(fbSegment_39);
fbSegment[40] := ADR(fbSegment_40);
fbSegment[41] := ADR(fbSegment_41);
fbSegment[42] := ADR(fbSegment_42);
fbSegment[43] := ADR(fbSegment_43);
fbSegment[44] := ADR(fbSegment_44);
fbSegment[45] := ADR(fbSegment_45);
fbSegment[46] := ADR(fbSegment_46);
fbSegment[47] := ADR(fbSegment_47);
END_ACTION

END_FUNCTION_BLOCK

// ---- MajorComponents/InterPlcComm/FB_ArbiterToSubSys_IO.TcPOU
(* Exchanges preemption requests and current beam state with subsystems in arbiter
network.

2019-12-2, A. Wallace

Use in conjunction with FB_SubSysToArbiter_IO.

This FB runs in the beamline arbiter PLC (BAP). There should be one of these for every
subsystem interfaced to the BAP. Each subsystem PLC should run a sibling FB_SubSysToArbiter_IO FB.

This FB and its subordinate communicate through the ethercat connection between the subsystem PLC and the BAP.

A beam parameter set request is sent from the subsystem to this PLC, and includes a cohort number.

This cohort number (i_RequestedBP.nCohortInt) is compared to a local cohort number (nRequestedCohort).
A request from the subsystem to update or modify its current request is indicated by an increase in the
i_RequestedBP.nCohortInt value. Then this function block updates the local arbiter request for the subsystem
and awaits confirmation. Once the new request is confirmed in the preemptive system this function block increments
the ActiveCohort value to match the nRequestedCohort. ActiveCohort is also relayed back to the subsystem
as the active cohort value in the o_CurrentBP set. The subsystem then knows its request has been heard,
and can carry out its own acknowledgement to its various requestors.

Things to note:
If a subsystem has any new or changed preemptive requests you should see the cohort value increment a bit.
If the cohort number is incrementing out of control, it usually means the subsysetm has some preemptive
request loop (two arbiters elevating to each other), or there is a RequestAdd, RequestRemove loop.

*)
FUNCTION_BLOCK FB_ArbiterToSubSys_IO
VAR_INPUT
    RequestingSystemID	:	DWORD := PMPS_GVL.EXCLUDED_ASSERTION_ID; // System ID for making requests to the supreme arbiter
    sName : STRING := 'ArbiterToSubSys';
    Reset : BOOL;
END_VAR
VAR_OUTPUT
END_VAR
VAR_IN_OUT
    Arbiter	: FB_Arbiter;
    fbFFHWO : FB_HardwareFFOutput;
END_VAR
VAR

    i_RequestedBP AT %I*	:	ST_BeamParams_IO; // Requested BP from subsystem
    {attribute 'pytmc' := '
        pv: RequestedBP:FromSubSys
    '}
    RequestedBP: ST_BeamParams;

    o_CurrentBP AT %Q* : ST_BeamParams_IO; // Current BP set

    // EL6692 Diagnostics
    i_Connected AT %I* : BOOL; // SYNC Inputs^External device not connected !!! Doesn't really work.
    {attribute 'pytmc' := 'pv: WcState
        io: i
        field: DESC Working counter state.
        field: ZNAM OK
        field: ONAM Error'}
    i_WcState AT %I* : BOOL := TRUE; // WcState^WcState
    {attribute 'pytmc' := 'pv: TxPDO_state
        io: i
        field: DESC PDO Transmission is OK
        field: ZNAM OK
        field: ONAM Error'}
    i_TxPDOState AT %I* : BOOL := TRUE; // SYNC Inputs^TxPDO state
    {attribute 'pytmc' := 'pv: TxPDO_toggle
        io: i
        field: DESC PDO Transmission is OK
        field: ZNAM OK
        field: ONAM Error'}
    i_TxPDOToggle AT %I* : BOOL; // TxPDO toggle

    // Fast faults
    ffPMPSIO_Disconnect : FB_FastFault := (i_Desc:='Issue w/ arbiter interface to subsystem, verify subsystem is OK, or ethercat connection.'); // Fast fault for ethercat issues
    nActiveCohort : UDINT := 0; // Active cohort. Updated to the req. number from the sub system after request is confirmed.
    nRequestedCohort : UDINT := 0;
    rtToggle : R_TRIG;
	fbToggleTimer : TON;
 	tInterval    : TIME := T#100mS;

END_VAR


// Incoming request from subsystem PLC
RequestedBP := IO_TO_BP(i_RequestedBP);

// Update Arbiter with our request
rtToggle(CLK:= i_RequestedBP.xValid); // If interface resumes, reset/catch up
// xValid will go false if the PLC program on the other side is stopped. Ironically the ethercat interface continues happily.
// If subsystem cohort has incremented, update beam parameter request with our arbiter
IF rtToggle.Q THEN
    nActiveCohort := 0;
END_IF

IF i_RequestedBP.nCohortInt > nRequestedCohort OR rtToggle.Q THEN
    Arbiter.RemoveRequest(RequestingSystemID);
    Arbiter.AddRequest(RequestingSystemID, RequestedBP,sName);
    nRequestedCohort := i_RequestedBP.nCohortInt;
END_IF


// Check if latest request is acknowledged by this arbiter
// Acknowledgement happens after an arbitration cycle, which means if RequestedCohort just incremented
// due to a new request, CheckRequest will be false.
IF Arbiter.CheckRequest(RequestingSystemID) THEN
    nActiveCohort := nRequestedCohort; // If it is, then the active cohort is set to the requested cohort number.
END_IF

fbToggleTimer(IN := NOT o_CurrentBP.xValidToggle, PT := tInterval);
// Sending current beam parameter set to subsystems
o_CurrentBP := BP_TO_IO(PMPS_GVL.stCurrentBeamParameters);
o_CurrentBP.nCohortInt := nActiveCohort;
IF (fbToggleTimer.Q) THEN o_CurrentBP.xValidToggle := NOT o_CurrentBP.xValidToggle; END_IF
o_CurrentBP.xValid := TRUE; // This is set and held true here every cycle to prove the PLC on this side is still running


//////////////////////////////////////
// Verifying the ethercat interface health
/////////////////////////////////////
// Both of these values should be 0 for a fully valid exchange
ffPMPSIO_Disconnect.i_xOK := NOT i_WcState AND NOT i_TxPDOState;

ffPMPSIO_Disconnect(
    io_fbFFHWO := fbFFHWO,
    i_xReset := Reset,
    i_DevName := sName,
    i_TypeCode:=5);

END_FUNCTION_BLOCK
